// TIA Portal V20 export
TYPE "typeWinderUseMode"
// stored: Access Published, IsFailsafeCompliant true, Namespace Safety
   STRUCT
      unwinderTopUse : Bool;
      unwinderBottomUse : Bool;
   END_STRUCT;
END_TYPE
